// TIA Portal V17 export
// export: Created 2023-04-07T15:18:38.2224118Z, ExportSetting WithDefaults, DisplayName Totally Integrated Automation Portal, DisplayVersion V17 Update 4, DisplayName TIA Portal Openness, DisplayVersion V17 Update 4, DisplayName TIA Portal Version Control Interface, DisplayVersion V17, DisplayName STEP 7 Professional, DisplayVersion V17 Update 4, DisplayName STEP 7 Safety, DisplayVersion V17, DisplayName WinCC Professional, DisplayVersion V17 Update 4
FUNCTION_BLOCK "State_Machine1"   // FB61, GRAPH
VERSION : 0.1
// stored: AcknowledgeErrorsRequired true, AutoNumber false, GraphVersion 6.0, InitialValuesAcquisition false, IsIECCheckEnabled false, LanguageInNetworks LAD, LockOperatingMode false, PermanentILProcessingInMANMode false, SetENOAutomatically false, SkipSteps false, UDAEnableTagReadback false, WithAlarmHandling true
   // inherited from GRAPH_BASE
   VAR
      OFF_SQ_BASE : Bool;
   END_VAR
   VAR_INPUT
      OFF_SQ { ExternalAccessible := 'False'; ExternalVisible := 'False'; ExternalWritable := 'False'} : Bool := false;   // Turn sequence off
      INIT_SQ { ExternalAccessible := 'False'; ExternalVisible := 'False'; ExternalWritable := 'False'} : Bool := false;   // Set sequence to initial state
      ACK_EF { ExternalAccessible := 'False'; ExternalVisible := 'False'; ExternalWritable := 'False'} : Bool := false;   // Acknowledge all errors and faults
      S_PREV { ExternalAccessible := 'False'; ExternalVisible := 'False'; ExternalWritable := 'False'} : Bool := false;   // Output previous step in parameter S_NO
      S_NEXT { ExternalAccessible := 'False'; ExternalVisible := 'False'; ExternalWritable := 'False'} : Bool := false;   // Indicate next step in parameter S_NO
      SW_AUTO { ExternalAccessible := 'False'; ExternalVisible := 'False'; ExternalWritable := 'False'} : Bool := false;   // Automatic mode
      SW_TAP { ExternalAccessible := 'False'; ExternalVisible := 'False'; ExternalWritable := 'False'} : Bool := false;   // Semiautomatic/switch with transition
      SW_TOP { ExternalAccessible := 'False'; ExternalVisible := 'False'; ExternalWritable := 'False'} : Bool := false;   // Semiautomatic/ignore transition
      SW_MAN { ExternalAccessible := 'False'; ExternalVisible := 'False'; ExternalWritable := 'False'} : Bool := false;   // Manual mode
      S_SEL { ExternalAccessible := 'False'; ExternalVisible := 'False'; ExternalWritable := 'False'} : Int := 0;   // Select step to be output to S_NO
      S_ON { ExternalAccessible := 'False'; ExternalVisible := 'False'; ExternalWritable := 'False'} : Bool := false;   // Activate step indicated in S_NO
      S_OFF { ExternalAccessible := 'False'; ExternalVisible := 'False'; ExternalWritable := 'False'} : Bool := false;   // Deactivate step indicated S_NO
      T_PUSH { ExternalAccessible := 'False'; ExternalVisible := 'False'; ExternalWritable := 'False'} : Bool := false;   // Enable transition to switch in semi automatic mode
   END_VAR
   VAR_OUTPUT
      S_NO { ExternalAccessible := 'False'; ExternalVisible := 'False'; ExternalWritable := 'False'} : Int := 0;   // Step number
      S_MORE { ExternalAccessible := 'False'; ExternalVisible := 'False'; ExternalWritable := 'False'} : Bool := false;   // More steps are available and can be shown in S_NO
      S_ACTIVE { ExternalAccessible := 'False'; ExternalVisible := 'False'; ExternalWritable := 'False'} : Bool := false;   // Step indicated in S_NO is active
      ERR_FLT { ExternalAccessible := 'False'; ExternalVisible := 'False'; ExternalWritable := 'False'} : Bool := false;   // Interlock or supervision group error
      AUTO_ON { ExternalAccessible := 'False'; ExternalVisible := 'False'; ExternalWritable := 'False'} : Bool := false;   // Automatic mode is active
      TAP_ON { ExternalAccessible := 'False'; ExternalVisible := 'False'; ExternalWritable := 'False'} : Bool := false;   // Semiautomatic mode/step with transition enabled
      TOP_ON { ExternalAccessible := 'False'; ExternalVisible := 'False'; ExternalWritable := 'False'} : Bool := false;   // Semiautomatic mode/ignore transition enabled
      MAN_ON { ExternalAccessible := 'False'; ExternalVisible := 'False'; ExternalWritable := 'False'} : Bool := false;   // Manual mode is active
   END_VAR
BEGIN
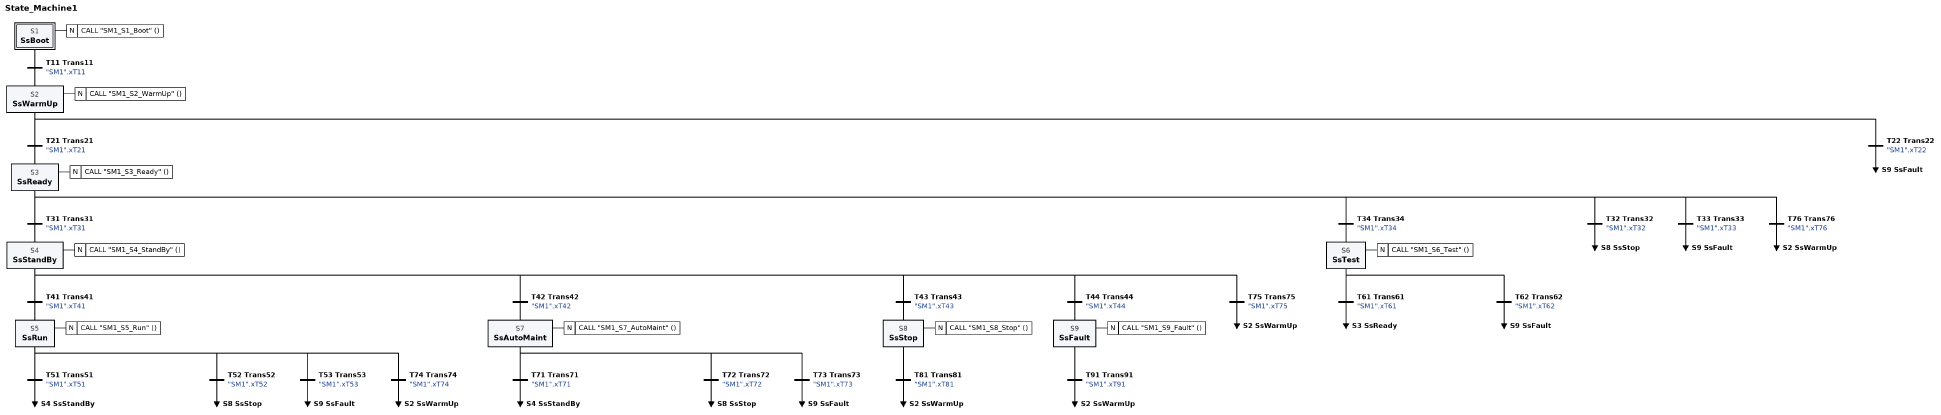
   // sequencer 1: State Machine Battery
   INITIAL_STEP SsBoot:   // S1, max time T#10S, warning time T#7S
              N    CALL "SM1_S1_Boot" ()
   END_STEP
   TRANSITION Trans11 FROM SsBoot TO SsWarmUp   // T11
      := "SM1".xT11;
   END_TRANSITION
   STEP SsWarmUp:   // S2, max time T#10S, warning time T#7S
              N    CALL "SM1_S2_WarmUp" ()
   END_STEP
   TRANSITION Trans21 FROM SsWarmUp TO SsReady   // T21
      := "SM1".xT21;
   END_TRANSITION
   TRANSITION Trans22 FROM SsWarmUp TO SsFault   // T22, jump
      := "SM1".xT22;
   END_TRANSITION
   STEP SsReady:   // S3, max time T#10S, warning time T#7S
              N    CALL "SM1_S3_Ready" ()
   END_STEP
   TRANSITION Trans31 FROM SsReady TO SsStandBy   // T31
      := "SM1".xT31;
   END_TRANSITION
   TRANSITION Trans34 FROM SsReady TO SsTest   // T34
      := "SM1".xT34;
   END_TRANSITION
   TRANSITION Trans32 FROM SsReady TO SsStop   // T32, jump
      := "SM1".xT32;
   END_TRANSITION
   TRANSITION Trans33 FROM SsReady TO SsFault   // T33, jump
      := "SM1".xT33;
   END_TRANSITION
   TRANSITION Trans76 FROM SsReady TO SsWarmUp   // T76, jump
      := "SM1".xT76;
   END_TRANSITION
   STEP SsStandBy:   // S4, max time T#10S, warning time T#7S
              N    CALL "SM1_S4_StandBy" ()
   END_STEP
   TRANSITION Trans41 FROM SsStandBy TO SsRun   // T41
      := "SM1".xT41;
   END_TRANSITION
   TRANSITION Trans42 FROM SsStandBy TO SsAutoMaint   // T42
      := "SM1".xT42;
   END_TRANSITION
   TRANSITION Trans43 FROM SsStandBy TO SsStop   // T43
      := "SM1".xT43;
   END_TRANSITION
   TRANSITION Trans44 FROM SsStandBy TO SsFault   // T44
      := "SM1".xT44;
   END_TRANSITION
   TRANSITION Trans75 FROM SsStandBy TO SsWarmUp   // T75, jump
      := "SM1".xT75;
   END_TRANSITION
   STEP SsRun:   // S5, max time T#10S, warning time T#7S
              N    CALL "SM1_S5_Run" ()
   END_STEP
   TRANSITION Trans51 FROM SsRun TO SsStandBy   // T51, jump
      := "SM1".xT51;
   END_TRANSITION
   TRANSITION Trans52 FROM SsRun TO SsStop   // T52, jump
      := "SM1".xT52;
   END_TRANSITION
   TRANSITION Trans53 FROM SsRun TO SsFault   // T53, jump
      := "SM1".xT53;
   END_TRANSITION
   TRANSITION Trans74 FROM SsRun TO SsWarmUp   // T74, jump
      := "SM1".xT74;
   END_TRANSITION
   STEP SsTest:   // S6, max time T#10S, warning time T#7S
              N    CALL "SM1_S6_Test" ()
   END_STEP
   TRANSITION Trans61 FROM SsTest TO SsReady   // T61, jump
      := "SM1".xT61;
   END_TRANSITION
   TRANSITION Trans62 FROM SsTest TO SsFault   // T62, jump
      := "SM1".xT62;
   END_TRANSITION
   STEP SsAutoMaint:   // S7, max time T#10S, warning time T#7S
              N    CALL "SM1_S7_AutoMaint" ()
   END_STEP
   TRANSITION Trans71 FROM SsAutoMaint TO SsStandBy   // T71, jump
      := "SM1".xT71;
   END_TRANSITION
   TRANSITION Trans72 FROM SsAutoMaint TO SsStop   // T72, jump
      := "SM1".xT72;
   END_TRANSITION
   TRANSITION Trans73 FROM SsAutoMaint TO SsFault   // T73, jump
      := "SM1".xT73;
   END_TRANSITION
   STEP SsStop:   // S8, max time T#10S, warning time T#7S
              N    CALL "SM1_S8_Stop" ()
   END_STEP
   TRANSITION Trans81 FROM SsStop TO SsWarmUp   // T81, jump
      := "SM1".xT81;
   END_TRANSITION
   STEP SsFault:   // S9, max time T#10S, warning time T#7S
              N    CALL "SM1_S9_Fault" ()
   END_STEP
   TRANSITION Trans91 FROM SsFault TO SsWarmUp   // T91, jump
      := "SM1".xT91;
   END_TRANSITION
END_FUNCTION_BLOCK
